Omron Sysmac Studio project ISA_T4Q5_b_1 (Sysmac Studio 1.23.0.14, StandardProject)

# Controller new_Controller_0: NX1P2-1040DT1 version 1.18
Task PrimaryTask (priority 4, period or condition 8000): Programa0
Library INV00x_MX2_ECT 1.0.9 (contents left out)

VAR_GLOBAL
    PP : BOOL;  (* Pulsador de Paro; at BuiltInIO://cpu/#0/Input_Bit_00 *)
    PM : BOOL;  (* Pulsador de Marcha; at BuiltInIO://cpu/#0/Input_Bit_01 *)
    PR : BOOL;  (* Pulsador de Reset; at BuiltInIO://cpu/#0/Input_Bit_02 *)
    Variador_01_Comando : WORD;  (* Comando del Variador 1; at ECAT://node#11/Command *)
    Variador_01_Frecuencia : UINT;  (* Consigna de frecuencia del Variador 1; at ECAT://node#11/Frequency reference *)
    presion_raw : INT;  (* Señal de presión de 4 a 20mA; at BuiltInIO://opt/#0/Ch1_Analog_Input_Value *)
    PP_HMI AT %W0.00 : BOOL;  (* Pulsador de Paro HMI; published *)
    PM_HMI AT %W0.01 : BOOL;  (* Pulsador de Marcha HMI; published *)
    PR_HMI AT %W0.02 : BOOL;  (* Pulsador de Reset HMI; published *)
END_VAR
VAR_GLOBAL RETAIN
    funcionamiento_motor_1 AT %D6 : REAL;  (* Porcentaje de funcionamiento motor 1; published *)
END_VAR
VAR_GLOBAL
    motor1_activo AT %W0.03 : BOOL;  (* Indicador motor 1 activo; published *)
    motor2_activo AT %W0.04 : BOOL;  (* Indicador motor 2 activo; published *)
END_VAR
VAR_GLOBAL RETAIN
    funcionamiento_motor_2 AT %D8 : REAL;  (* Porcentaje de funcionamiento motor 2; published *)
    presion_real AT %D0 : REAL;  (* Presión del tanque en bares; published *)
    caudal_1_real AT %D2 : REAL;  (* Caudal del motor 1 en m_3/min; published *)
END_VAR
VAR_GLOBAL
    Variador_02_Comando : WORD;  (* Comando del Variador 2; at ECAT://node#5/Command *)
    Variador_02_Frecuencia : UINT;  (* Consigna de Frecuencia del Variador 2; at ECAT://node#5/Frequency reference *)
END_VAR
VAR_GLOBAL RETAIN
    caudal_2_real AT %D4 : REAL;  (* Caudal del motor 2 en m_3/min; published *)
END_VAR

PROGRAM Programa0
VAR
    presion_limitada_m1 : REAL;  (* Presion limitada de 30 a 45 bar *)
    presion_limitada_m2 : REAL;  (* Presion limitada de 10 a 30 bar *)
END_VAR
VAR CONSTANT
    caudal_referencia : REAL := 0.5;  (* Caudal de referencia para cálculos *)
    frecuencia_referencia : REAL := 50;  (* Frecuencia de referencia para cálculos *)
END_VAR
VAR
    frecuencia_1_real : REAL;  (* Frecuencia de giro real del motor 1 *)
    frecuencia_2_real : REAL;  (* Frecuencia de giro real del motor 2 *)
    presion_raw_limitada : INT;  (* Señal de presion limitada a [400..2000] *)
    Reset : ResetECError;
    Busy : BOOL;
    Error : BOOL;  (* Sistema en error *)
    Error_ID : WORD;  (* Identificador de error *)
    PR_VAR : BOOL;  (* Variable del Pulsador de Reset *)
    PP_VAR : BOOL;  (* Variable del Pulsador de Paro *)
    PM_VAR : BOOL;  (* Variable del Pulsador de Marcha *)
    sistema_activo : BOOL := False;  (* Indicador de sistema funcionando o no *)
END_VAR
VAR_EXTERNAL
    PM : BOOL;  (* Pulsador de Marcha *)
    Variador_01_Comando : WORD;  (* Comando del variador 1 *)
    PP : BOOL;  (* Pulsador de Paro *)
    Variador_01_Frecuencia : UINT;
    presion_raw : INT;
    PM_HMI : BOOL;
    presion_real : REAL;
    caudal_1_real : REAL;
    Variador_02_Comando : WORD;
    caudal_2_real : REAL;
    Variador_02_Frecuencia : UINT;
    PR : BOOL;
    PR_HMI : BOOL;
    PP_HMI : BOOL;
    funcionamiento_motor_2 : REAL;
    funcionamiento_motor_1 : REAL;
    motor2_activo : BOOL;
    motor1_activo : BOOL;
END_VAR

(* Section calculos: ladder, written here as Structured Text *)

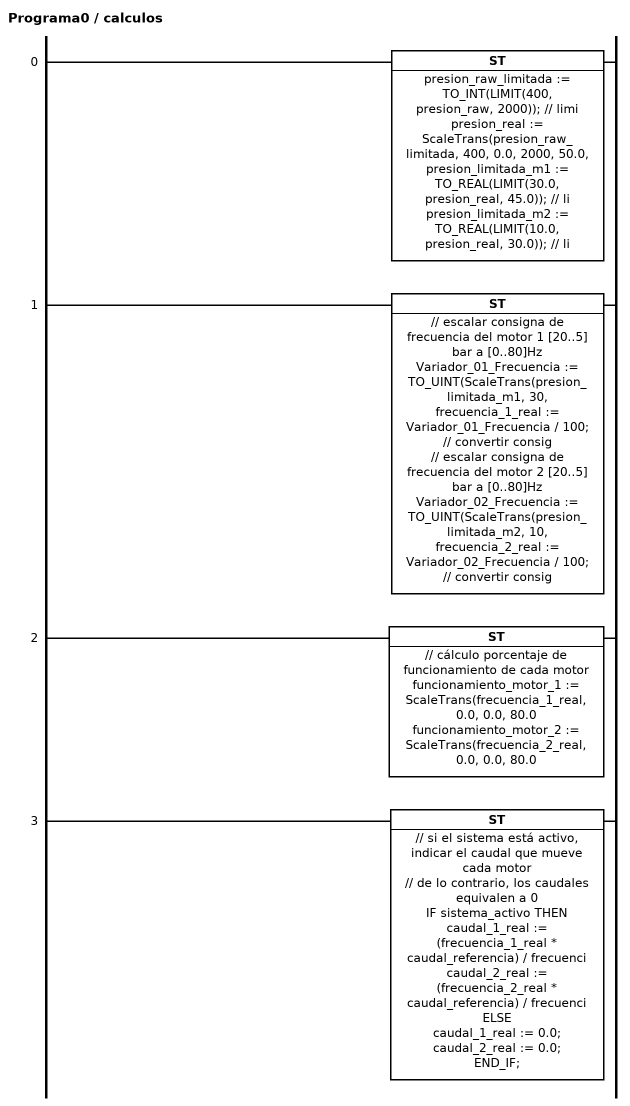
(* Rung 0 *)
presion_raw_limitada := TO_INT(LIMIT(400, presion_raw, 2000)); // limitación previa de [0..20]mA a [4..20]mA
presion_real := ScaleTrans(presion_raw_limitada, 400, 0.0, 2000, 50.0, 0.0); // escalar a [0..25]bar
presion_limitada_m1 := TO_REAL(LIMIT(30.0, presion_real, 45.0)); // limitar presión de [0..25] a [30..45] bar
presion_limitada_m2 := TO_REAL(LIMIT(10.0, presion_real, 30.0)); // limitar presión de [0..25] a [10..30] bar
(* Rung 1 *)
// escalar consigna de frecuencia del motor 1 [20..5] bar a [0..80]Hz
Variador_01_Frecuencia := TO_UINT(ScaleTrans(presion_limitada_m1, 30, 8000, 45, 0, 0));
frecuencia_1_real := Variador_01_Frecuencia / 100; // convertir consigna para visualizar con dos decimales

// escalar consigna de frecuencia del motor 2 [20..5] bar a [0..80]Hz
Variador_02_Frecuencia := TO_UINT(ScaleTrans(presion_limitada_m2, 10, 8000, 30, 0, 0));
frecuencia_2_real := Variador_02_Frecuencia / 100; // convertir consigna para visualizar con dos decimales
(* Rung 2 *)
// cálculo porcentaje de funcionamiento de cada motor
funcionamiento_motor_1 := ScaleTrans(frecuencia_1_real, 0.0, 0.0, 80.0, 100.0, 0);
funcionamiento_motor_2 := ScaleTrans(frecuencia_2_real, 0.0, 0.0, 80.0, 100.0, 0);
(* Rung 3 *)
// si el sistema está activo, indicar el caudal que mueve cada motor
// de lo contrario, los caudales equivalen a 0
IF sistema_activo THEN
	caudal_1_real := (frecuencia_1_real * caudal_referencia) / frecuencia_referencia;
	caudal_2_real := (frecuencia_2_real * caudal_referencia) / frecuencia_referencia;
ELSE
	caudal_1_real := 0.0;
	caudal_2_real := 0.0;
END_IF;

(* Section principal: ladder, written here as Structured Text *)

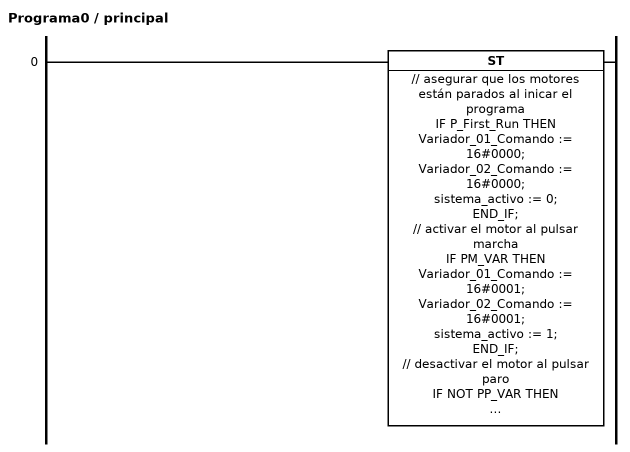
(* Rung 0 *)
// asegurar que los motores están parados al inicar el programa
IF P_First_Run THEN
	Variador_01_Comando := 16#0000;
	Variador_02_Comando := 16#0000;
	sistema_activo := 0;
END_IF;

// activar el motor al pulsar marcha
IF PM_VAR THEN
	Variador_01_Comando := 16#0001;
	Variador_02_Comando := 16#0001;
	sistema_activo := 1;
END_IF;

// desactivar el motor al pulsar paro
IF NOT PP_VAR THEN
	Variador_01_Comando := 16#0000;
	Variador_02_Comando := 16#0000;
	sistema_activo := 0;
END_IF;

(* Section hmi_plc: ladder, written here as Structured Text *)

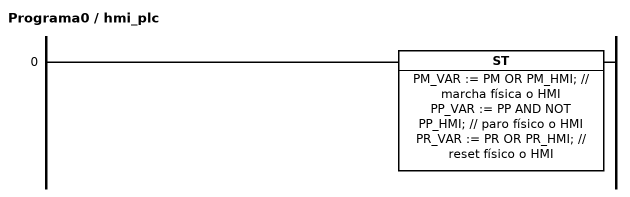
(* Rung 0 *)
PM_VAR := PM OR PM_HMI; // marcha física o HMI
PP_VAR := PP AND NOT PP_HMI; // paro físico o HMI
PR_VAR := PR OR PR_HMI; // reset físico o HMI

(* Section reset: ladder, written here as Structured Text *)

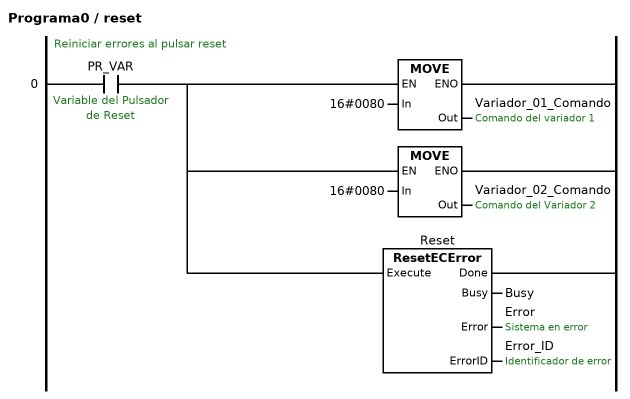
(* Rung 0: Reiniciar errores al pulsar reset *)
IF PR_VAR THEN
    Variador_01_Comando := 16#0080;
    Variador_02_Comando := 16#0080;
END_IF;
Reset(Execute := PR_VAR, Busy => Busy, Error => Error, ErrorID => Error_ID);

(* Section movimiento: ladder, written here as Structured Text *)

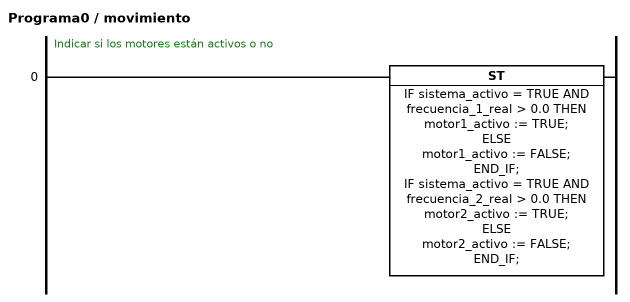
(* Rung 0: Indicar si los motores están activos o no *)
IF sistema_activo = TRUE AND frecuencia_1_real > 0.0 THEN
	motor1_activo := TRUE;
ELSE
	motor1_activo := FALSE;
END_IF;

IF sistema_activo = TRUE AND frecuencia_2_real > 0.0 THEN
	motor2_activo := TRUE;
ELSE
	motor2_activo := FALSE;
END_IF;
END_PROGRAM